KUKA KRL program: MOD.src

&ACCESS RV1
&REL 2
&PARAM TEMPLATE = C:\KRC\Roboter\Template\FunctionVorgabe
&PARAM EDITMASK = *
DEFFCT REAL MOD(RV1:IN, RV2:IN)
  REAL RV1, RV2
  REAL RET_VAL
  INT TEMP

  TEMP = WHOLE(RV1 / RV2)
  RET_VAL = RV1 - (RV2 * TEMP)

  RETURN(RET_VAL)
ENDFCT
